(* Logix 5000 project; controller R1USB70001_CWRU_Scenario_Gen_20111116 vendor 1 type 14 code 54 rev 19.11; software revision 19.01; part 3 of 9 *)
(* tags used below, declared in another part *)
   DiscreteOutputsPv : DiscreteOutputsPv;
   EditScenarioPv : EditScenarioPv;
   CL_LP_B1_L1_SG1 : ALIAS FOR ACNR_CP_SG_N5:1:O.2;
   CL_LP_B1_L1_SG2 : ALIAS FOR ACNR_CP_SG_N5:1:O.3;
   CL_LP_B1_L2_SG1 : ALIAS FOR ACNR_CP_SG_N5:1:O.4;
   CL_LP_B1_L2_SG2 : ALIAS FOR ACNR_CP_SG_N5:1:O.5;
   CL_LP_B1_L3_SG1 : ALIAS FOR ACNR_CP_SG_N5:1:O.6;
   CL_LP_B1_L3_SG2 : ALIAS FOR ACNR_CP_SG_N5:1:O.7;
   CL_LP_B1_L4_SG1 : ALIAS FOR ACNR_CP_SG_N5:2:O.0;
   CL_LP_B1_L4_SG2 : ALIAS FOR ACNR_CP_SG_N5:2:O.1;
   CL_LP_B1_L5_SG1 : ALIAS FOR ACNR_CP_SG_N5:2:O.2;
   CL_LP_B1_L5_SG2 : ALIAS FOR ACNR_CP_SG_N5:2:O.3;
   CL_LP_B1_SG : ALIAS FOR ACNR_CP_SG_N5:1:O.1;
   CL_LP_B2_L1_SG1 : ALIAS FOR ACNR_CP_SG_N5:2:O.5;
   CL_LP_B2_L1_SG2 : ALIAS FOR ACNR_CP_SG_N5:2:O.6;
   CL_LP_B2_L2_SG1 : ALIAS FOR ACNR_CP_SG_N5:3:O.0;
   CL_LP_B2_L2_SG2 : ALIAS FOR ACNR_CP_SG_N5:3:O.1;
   CL_LP_B2_L3_SG1 : ALIAS FOR ACNR_CP_SG_N5:3:O.2;
   CL_LP_B2_L3_SG2 : ALIAS FOR ACNR_CP_SG_N5:3:O.3;
   CL_LP_B2_L4_SG1 : ALIAS FOR ACNR_CP_SG_N5:3:O.4;
   CL_LP_B2_L4_SG2 : ALIAS FOR ACNR_CP_SG_N5:3:O.5;
   CL_LP_B2_L5_SG1 : ALIAS FOR ACNR_CP_SG_N5:3:O.6;
   CL_LP_B2_L5_SG2 : ALIAS FOR ACNR_CP_SG_N5:3:O.7;
   CL_LP_B2_SG : ALIAS FOR ACNR_CP_SG_N5:2:O.4;
   CL_LP_ML_SG : ALIAS FOR ACNR_CP_SG_N5:1:O.0;
   EditScenario : EditScenarioPub;
   HMI : HMIPub;
   IL_LP_B1_L1_SG1 : ALIAS FOR ACNR_CP_SG_N5:4:O.2;
   IL_LP_B1_L1_SG2 : ALIAS FOR ACNR_CP_SG_N5:4:O.3;
   IL_LP_B1_L2_SG1 : ALIAS FOR ACNR_CP_SG_N5:4:O.4;
   IL_LP_B1_L2_SG2 : ALIAS FOR ACNR_CP_SG_N5:4:O.5;
   IL_LP_B1_L3_SG1 : ALIAS FOR ACNR_CP_SG_N5:4:O.6;
   IL_LP_B1_L3_SG2 : ALIAS FOR ACNR_CP_SG_N5:4:O.7;
   IL_LP_B1_L4_SG1 : ALIAS FOR ACNR_CP_SG_N5:5:O.0;
   IL_LP_B1_L4_SG2 : ALIAS FOR ACNR_CP_SG_N5:5:O.1;
   IL_LP_B1_L5_SG1 : ALIAS FOR ACNR_CP_SG_N5:5:O.2;
   IL_LP_B1_L5_SG2 : ALIAS FOR ACNR_CP_SG_N5:5:O.3;
   IL_LP_B1_SG : ALIAS FOR ACNR_CP_SG_N5:4:O.1;
   IL_LP_B2_L1_SG1 : ALIAS FOR ACNR_CP_SG_N5:5:O.5;
   IL_LP_B2_L1_SG2 : ALIAS FOR ACNR_CP_SG_N5:5:O.6;
   IL_LP_B2_L2_SG1 : ALIAS FOR ACNR_CP_SG_N5:6:O.0;
   IL_LP_B2_L2_SG2 : ALIAS FOR ACNR_CP_SG_N5:6:O.1;
   IL_LP_B2_L3_SG1 : ALIAS FOR ACNR_CP_SG_N5:6:O.2;
   IL_LP_B2_L3_SG2 : ALIAS FOR ACNR_CP_SG_N5:6:O.3;
   IL_LP_B2_L4_SG1 : ALIAS FOR ACNR_CP_SG_N5:6:O.4;
   IL_LP_B2_L4_SG2 : ALIAS FOR ACNR_CP_SG_N5:6:O.5;
   IL_LP_B2_L5_SG1 : ALIAS FOR ACNR_CP_SG_N5:6:O.6;
   IL_LP_B2_L5_SG2 : ALIAS FOR ACNR_CP_SG_N5:6:O.7;
   IL_LP_B2_SG : ALIAS FOR ACNR_CP_SG_N5:5:O.4;
   IL_LP_ML_SG : ALIAS FOR ACNR_CP_SG_N5:4:O.0;
   RL_LP_B1_L5_SG2 : ALIAS FOR ACNR_RP_SG_N4:2:O.3;
   RL_LP_B2_L1_SG1 : ALIAS FOR ACNR_RP_SG_N4:2:O.5;
   RL_LP_B2_L1_SG2 : ALIAS FOR ACNR_RP_SG_N4:2:O.6;
   RL_LP_B2_L2_SG1 : ALIAS FOR ACNR_RP_SG_N4:2:O.7;
   RL_LP_B2_L2_SG2 : ALIAS FOR ACNR_RP_SG_N4:3:O.0;
   RL_LP_B2_L3_SG1 : ALIAS FOR ACNR_RP_SG_N4:3:O.1;
   RL_LP_B2_L3_SG2 : ALIAS FOR ACNR_RP_SG_N4:3:O.2;
   RL_LP_B2_L4_SG1 : ALIAS FOR ACNR_RP_SG_N4:3:O.3;
   RL_LP_B2_L4_SG2 : ALIAS FOR ACNR_RP_SG_N4:3:O.4;
   RL_LP_B2_L5_SG1 : ALIAS FOR ACNR_RP_SG_N4:3:O.5;
   RL_LP_B2_L5_SG2 : ALIAS FOR ACNR_RP_SG_N4:3:O.6;
   RL_LP_B2_SG : ALIAS FOR ACNR_RP_SG_N4:2:O.4;
   RL_LP_B3_L1_SG1 : ALIAS FOR ACNR_RP_SG_N4:4:O.0;
   RL_LP_B3_L1_SG2 : ALIAS FOR ACNR_RP_SG_N4:4:O.1;
   RL_LP_B3_L2_SG1 : ALIAS FOR ACNR_RP_SG_N4:4:O.2;
   RL_LP_B3_L2_SG2 : ALIAS FOR ACNR_RP_SG_N4:4:O.3;
   RL_LP_B3_L3_SG1 : ALIAS FOR ACNR_RP_SG_N4:4:O.4;
   RL_LP_B3_L3_SG2 : ALIAS FOR ACNR_RP_SG_N4:4:O.5;
   RL_LP_B3_L4_SG1 : ALIAS FOR ACNR_RP_SG_N4:4:O.6;
   RL_LP_B3_L4_SG2 : ALIAS FOR ACNR_RP_SG_N4:4:O.7;
   RL_LP_B3_L5_SG1 : ALIAS FOR ACNR_RP_SG_N4:5:O.0;
   RL_LP_B3_L5_SG2 : ALIAS FOR ACNR_RP_SG_N4:5:O.1;
   RL_LP_B3_SG : ALIAS FOR ACNR_RP_SG_N4:3:O.7;
   RL_LP_B4_L1_SG1 : ALIAS FOR ACNR_RP_SG_N4:5:O.3;
   RL_LP_B4_L1_SG2 : ALIAS FOR ACNR_RP_SG_N4:5:O.4;
   RL_LP_B4_L2_SG1 : ALIAS FOR ACNR_RP_SG_N4:5:O.5;
   RL_LP_B4_L2_SG2 : ALIAS FOR ACNR_RP_SG_N4:5:O.6;
   RL_LP_B4_L3_SG1 : ALIAS FOR ACNR_RP_SG_N4:5:O.7;
   RL_LP_B4_L3_SG2 : ALIAS FOR ACNR_RP_SG_N4:6:O.0;
   RL_LP_B4_L4_SG1 : ALIAS FOR ACNR_RP_SG_N4:6:O.1;
   RL_LP_B4_L4_SG2 : ALIAS FOR ACNR_RP_SG_N4:6:O.2;
   RL_LP_B4_L5_SG1 : ALIAS FOR ACNR_RP_SG_N4:6:O.3;
   RL_LP_B4_L5_SG2 : ALIAS FOR ACNR_RP_SG_N4:6:O.4;
   RL_LP_B4_SG : ALIAS FOR ACNR_RP_SG_N4:5:O.2;
   Scenario : Scenario_Def[100];
(* MainProgram, continued *)

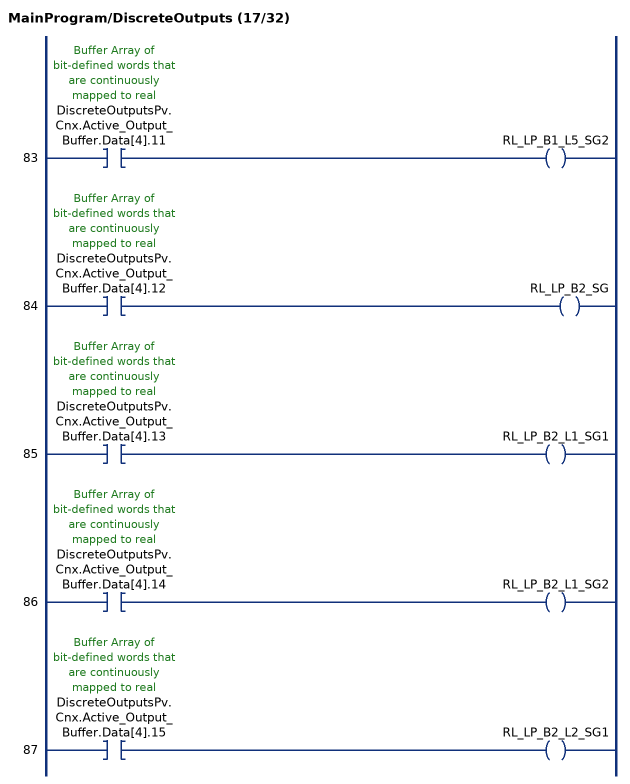
   83: XIC(DiscreteOutputsPv.Cnx.Active_Output_Buffer.Data[4].11)OTE(RL_LP_B1_L5_SG2);
   84: XIC(DiscreteOutputsPv.Cnx.Active_Output_Buffer.Data[4].12)OTE(RL_LP_B2_SG);
   85: XIC(DiscreteOutputsPv.Cnx.Active_Output_Buffer.Data[4].13)OTE(RL_LP_B2_L1_SG1);
   86: XIC(DiscreteOutputsPv.Cnx.Active_Output_Buffer.Data[4].14)OTE(RL_LP_B2_L1_SG2);
   87: XIC(DiscreteOutputsPv.Cnx.Active_Output_Buffer.Data[4].15)OTE(RL_LP_B2_L2_SG1);
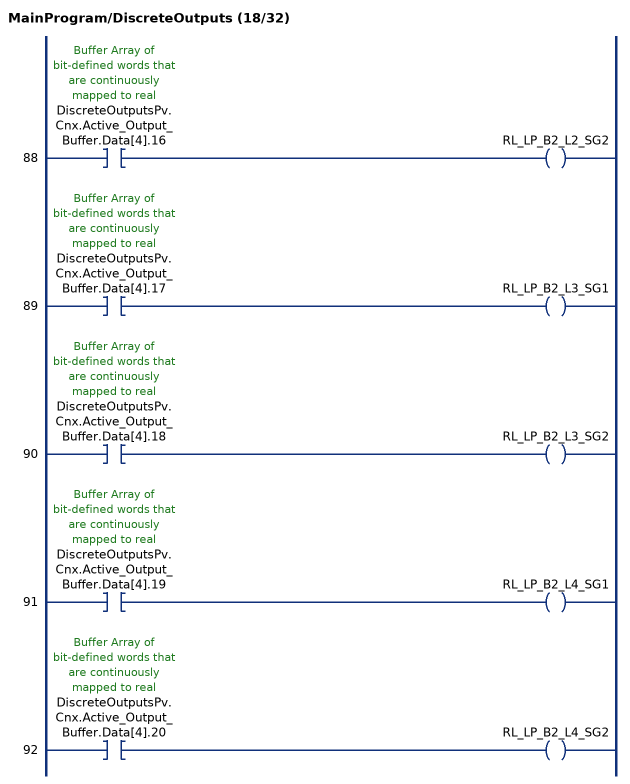
   88: XIC(DiscreteOutputsPv.Cnx.Active_Output_Buffer.Data[4].16)OTE(RL_LP_B2_L2_SG2);
   89: XIC(DiscreteOutputsPv.Cnx.Active_Output_Buffer.Data[4].17)OTE(RL_LP_B2_L3_SG1);
   90: XIC(DiscreteOutputsPv.Cnx.Active_Output_Buffer.Data[4].18)OTE(RL_LP_B2_L3_SG2);
   91: XIC(DiscreteOutputsPv.Cnx.Active_Output_Buffer.Data[4].19)OTE(RL_LP_B2_L4_SG1);
   92: XIC(DiscreteOutputsPv.Cnx.Active_Output_Buffer.Data[4].20)OTE(RL_LP_B2_L4_SG2);
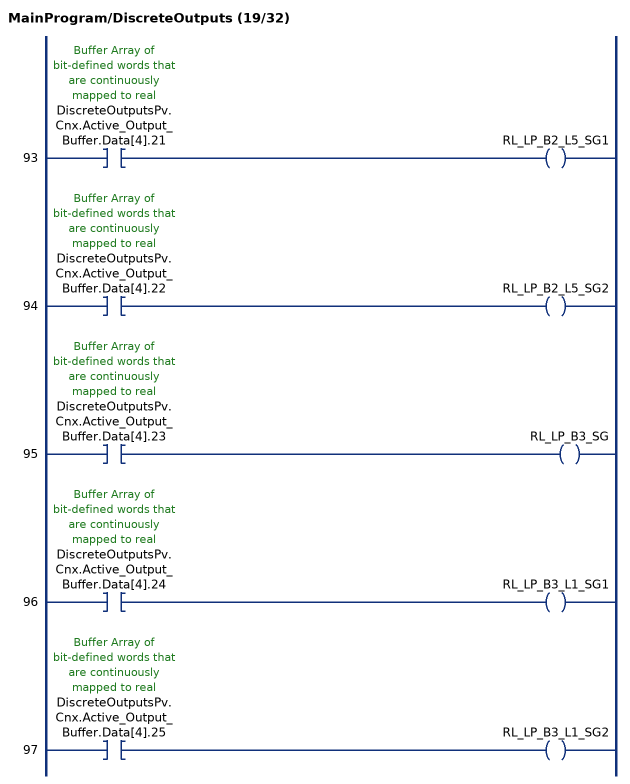
   93: XIC(DiscreteOutputsPv.Cnx.Active_Output_Buffer.Data[4].21)OTE(RL_LP_B2_L5_SG1);
   94: XIC(DiscreteOutputsPv.Cnx.Active_Output_Buffer.Data[4].22)OTE(RL_LP_B2_L5_SG2);
   95: XIC(DiscreteOutputsPv.Cnx.Active_Output_Buffer.Data[4].23)OTE(RL_LP_B3_SG);
   96: XIC(DiscreteOutputsPv.Cnx.Active_Output_Buffer.Data[4].24)OTE(RL_LP_B3_L1_SG1);
   97: XIC(DiscreteOutputsPv.Cnx.Active_Output_Buffer.Data[4].25)OTE(RL_LP_B3_L1_SG2);
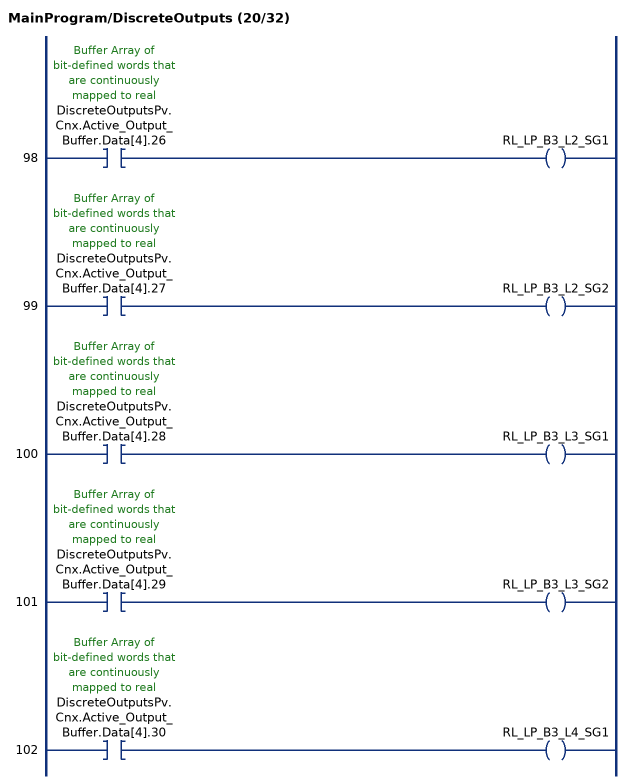
   98: XIC(DiscreteOutputsPv.Cnx.Active_Output_Buffer.Data[4].26)OTE(RL_LP_B3_L2_SG1);
   99: XIC(DiscreteOutputsPv.Cnx.Active_Output_Buffer.Data[4].27)OTE(RL_LP_B3_L2_SG2);
   100: XIC(DiscreteOutputsPv.Cnx.Active_Output_Buffer.Data[4].28)OTE(RL_LP_B3_L3_SG1);
   101: XIC(DiscreteOutputsPv.Cnx.Active_Output_Buffer.Data[4].29)OTE(RL_LP_B3_L3_SG2);
   102: XIC(DiscreteOutputsPv.Cnx.Active_Output_Buffer.Data[4].30)OTE(RL_LP_B3_L4_SG1);
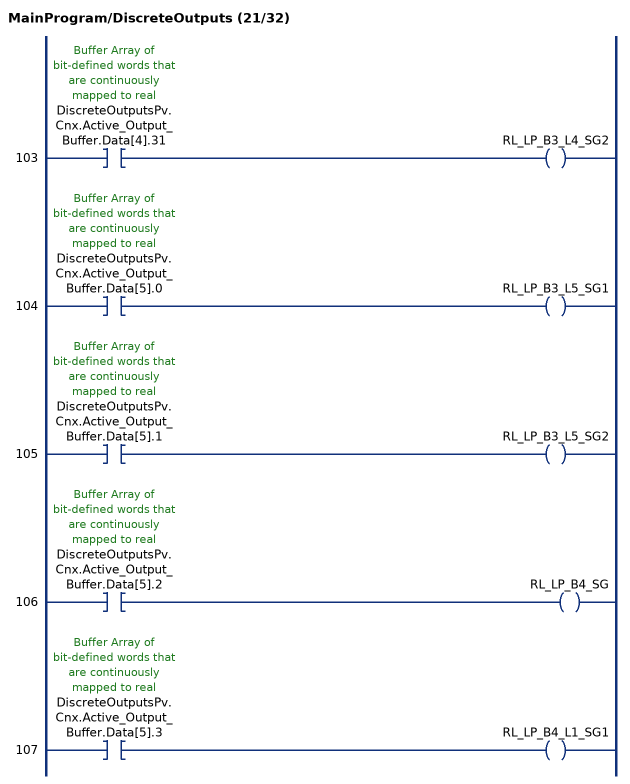
   103: XIC(DiscreteOutputsPv.Cnx.Active_Output_Buffer.Data[4].31)OTE(RL_LP_B3_L4_SG2);
   104: XIC(DiscreteOutputsPv.Cnx.Active_Output_Buffer.Data[5].0)OTE(RL_LP_B3_L5_SG1);
   105: XIC(DiscreteOutputsPv.Cnx.Active_Output_Buffer.Data[5].1)OTE(RL_LP_B3_L5_SG2);
   106: XIC(DiscreteOutputsPv.Cnx.Active_Output_Buffer.Data[5].2)OTE(RL_LP_B4_SG);
   107: XIC(DiscreteOutputsPv.Cnx.Active_Output_Buffer.Data[5].3)OTE(RL_LP_B4_L1_SG1);
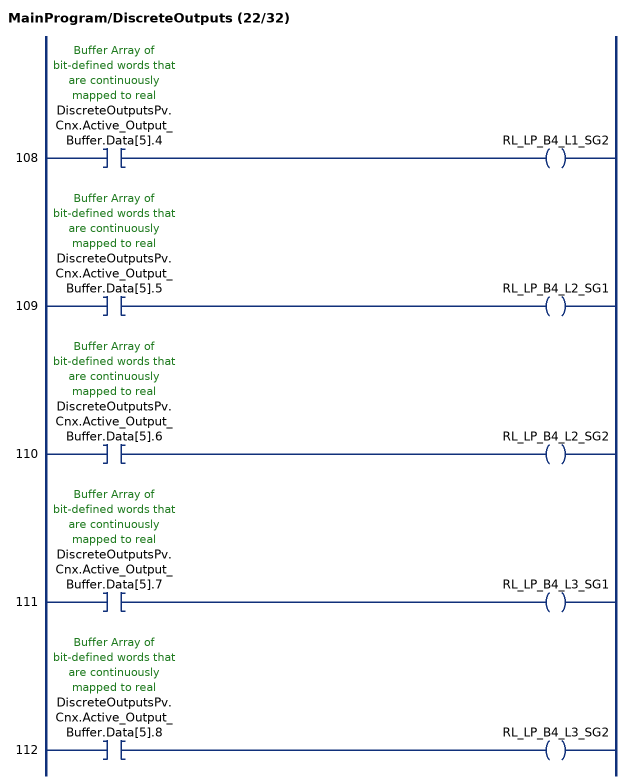
   108: XIC(DiscreteOutputsPv.Cnx.Active_Output_Buffer.Data[5].4)OTE(RL_LP_B4_L1_SG2);
   109: XIC(DiscreteOutputsPv.Cnx.Active_Output_Buffer.Data[5].5)OTE(RL_LP_B4_L2_SG1);
   110: XIC(DiscreteOutputsPv.Cnx.Active_Output_Buffer.Data[5].6)OTE(RL_LP_B4_L2_SG2);
   111: XIC(DiscreteOutputsPv.Cnx.Active_Output_Buffer.Data[5].7)OTE(RL_LP_B4_L3_SG1);
   112: XIC(DiscreteOutputsPv.Cnx.Active_Output_Buffer.Data[5].8)OTE(RL_LP_B4_L3_SG2);
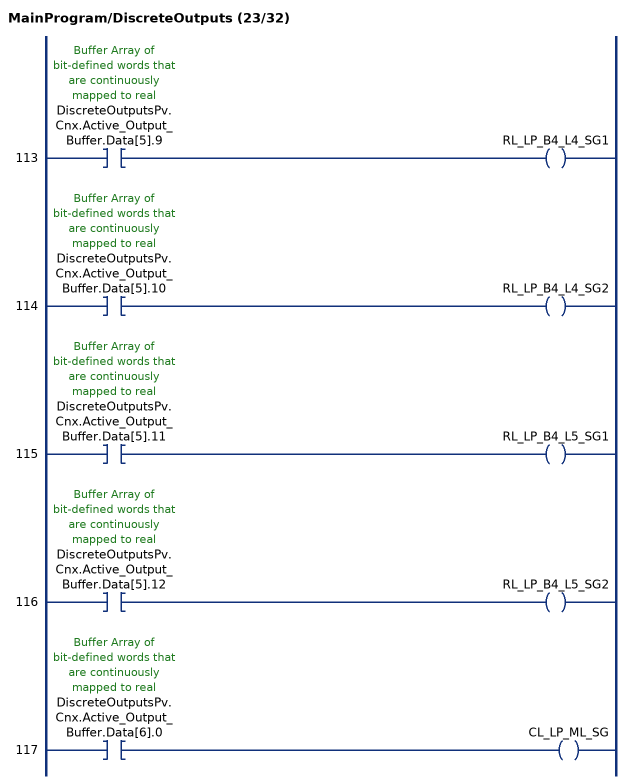
   113: XIC(DiscreteOutputsPv.Cnx.Active_Output_Buffer.Data[5].9)OTE(RL_LP_B4_L4_SG1);
   114: XIC(DiscreteOutputsPv.Cnx.Active_Output_Buffer.Data[5].10)OTE(RL_LP_B4_L4_SG2);
   115: XIC(DiscreteOutputsPv.Cnx.Active_Output_Buffer.Data[5].11)OTE(RL_LP_B4_L5_SG1);
   116: XIC(DiscreteOutputsPv.Cnx.Active_Output_Buffer.Data[5].12)OTE(RL_LP_B4_L5_SG2);
   117: XIC(DiscreteOutputsPv.Cnx.Active_Output_Buffer.Data[6].0)OTE(CL_LP_ML_SG);
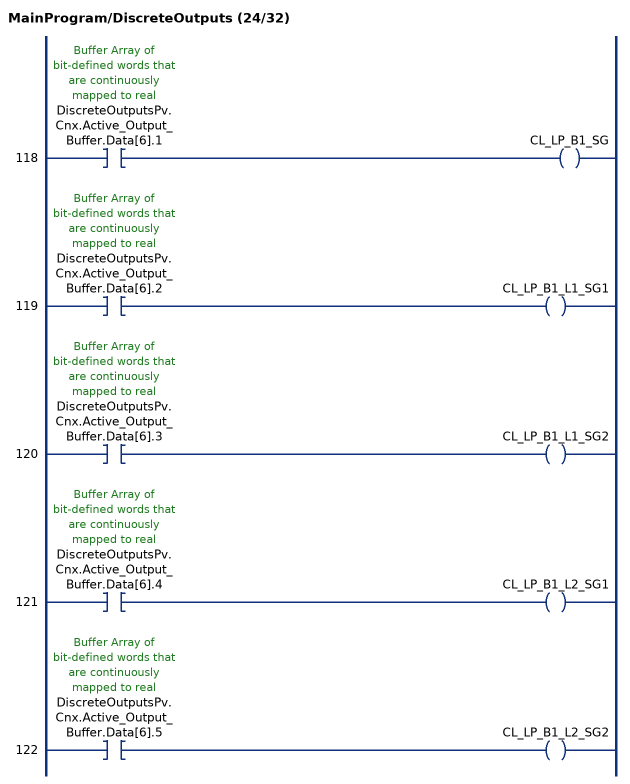
   118: XIC(DiscreteOutputsPv.Cnx.Active_Output_Buffer.Data[6].1)OTE(CL_LP_B1_SG);
   119: XIC(DiscreteOutputsPv.Cnx.Active_Output_Buffer.Data[6].2)OTE(CL_LP_B1_L1_SG1);
   120: XIC(DiscreteOutputsPv.Cnx.Active_Output_Buffer.Data[6].3)OTE(CL_LP_B1_L1_SG2);
   121: XIC(DiscreteOutputsPv.Cnx.Active_Output_Buffer.Data[6].4)OTE(CL_LP_B1_L2_SG1);
   122: XIC(DiscreteOutputsPv.Cnx.Active_Output_Buffer.Data[6].5)OTE(CL_LP_B1_L2_SG2);
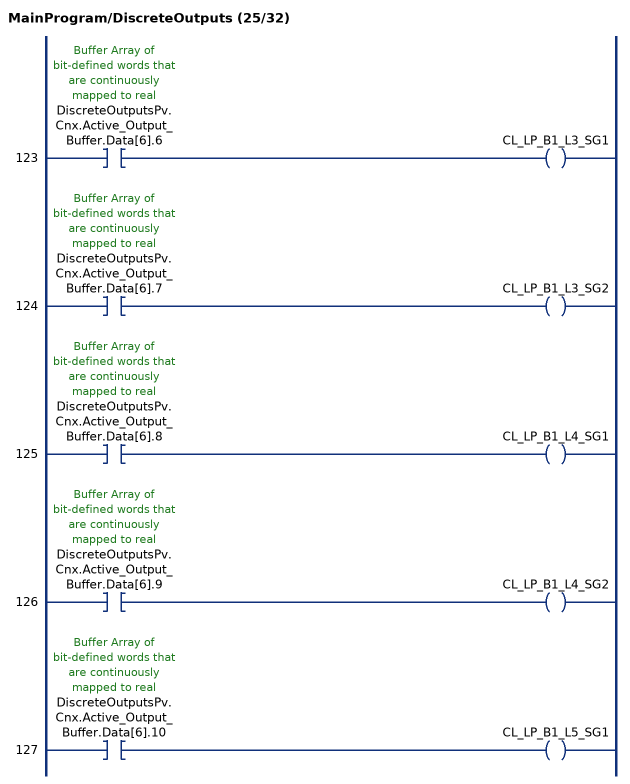
   123: XIC(DiscreteOutputsPv.Cnx.Active_Output_Buffer.Data[6].6)OTE(CL_LP_B1_L3_SG1);
   124: XIC(DiscreteOutputsPv.Cnx.Active_Output_Buffer.Data[6].7)OTE(CL_LP_B1_L3_SG2);
   125: XIC(DiscreteOutputsPv.Cnx.Active_Output_Buffer.Data[6].8)OTE(CL_LP_B1_L4_SG1);
   126: XIC(DiscreteOutputsPv.Cnx.Active_Output_Buffer.Data[6].9)OTE(CL_LP_B1_L4_SG2);
   127: XIC(DiscreteOutputsPv.Cnx.Active_Output_Buffer.Data[6].10)OTE(CL_LP_B1_L5_SG1);
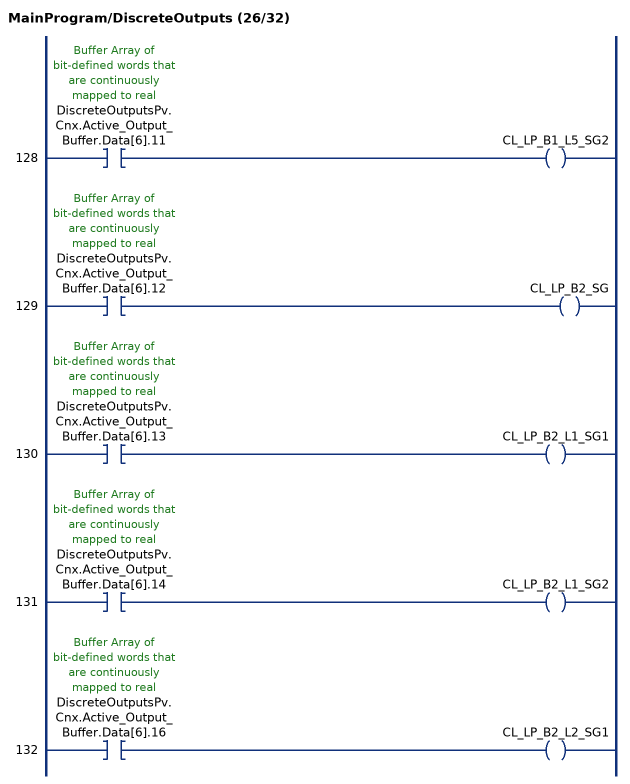
   128: XIC(DiscreteOutputsPv.Cnx.Active_Output_Buffer.Data[6].11)OTE(CL_LP_B1_L5_SG2);
   129: XIC(DiscreteOutputsPv.Cnx.Active_Output_Buffer.Data[6].12)OTE(CL_LP_B2_SG);
   130: XIC(DiscreteOutputsPv.Cnx.Active_Output_Buffer.Data[6].13)OTE(CL_LP_B2_L1_SG1);
   131: XIC(DiscreteOutputsPv.Cnx.Active_Output_Buffer.Data[6].14)OTE(CL_LP_B2_L1_SG2);
   132: XIC(DiscreteOutputsPv.Cnx.Active_Output_Buffer.Data[6].16)OTE(CL_LP_B2_L2_SG1);
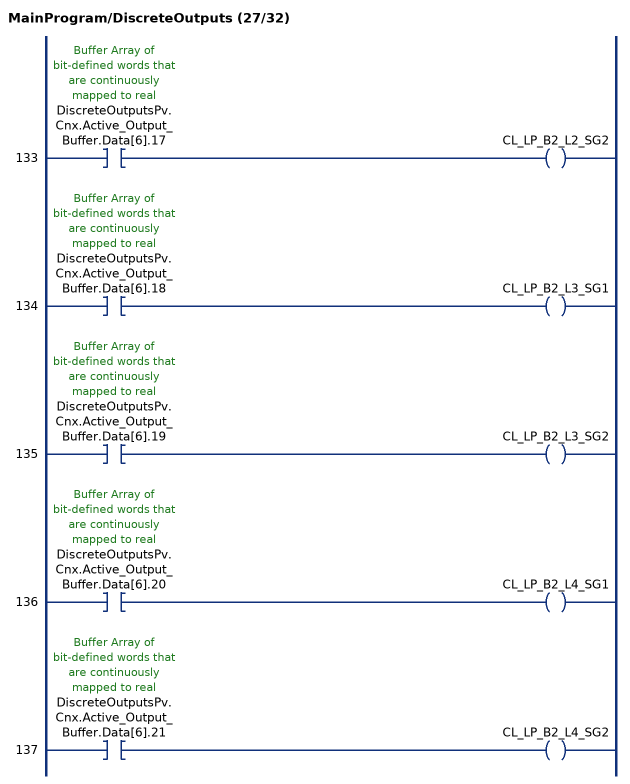
   133: XIC(DiscreteOutputsPv.Cnx.Active_Output_Buffer.Data[6].17)OTE(CL_LP_B2_L2_SG2);
   134: XIC(DiscreteOutputsPv.Cnx.Active_Output_Buffer.Data[6].18)OTE(CL_LP_B2_L3_SG1);
   135: XIC(DiscreteOutputsPv.Cnx.Active_Output_Buffer.Data[6].19)OTE(CL_LP_B2_L3_SG2);
   136: XIC(DiscreteOutputsPv.Cnx.Active_Output_Buffer.Data[6].20)OTE(CL_LP_B2_L4_SG1);
   137: XIC(DiscreteOutputsPv.Cnx.Active_Output_Buffer.Data[6].21)OTE(CL_LP_B2_L4_SG2);
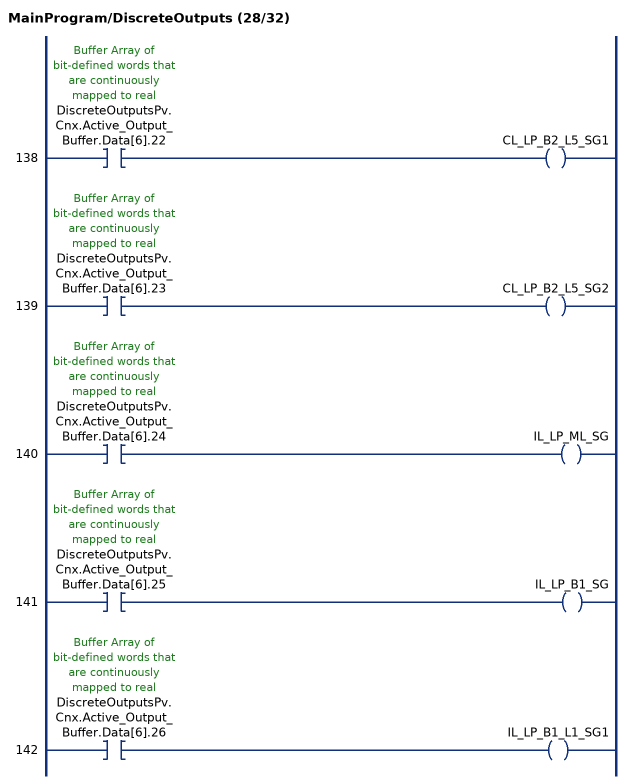
   138: XIC(DiscreteOutputsPv.Cnx.Active_Output_Buffer.Data[6].22)OTE(CL_LP_B2_L5_SG1);
   139: XIC(DiscreteOutputsPv.Cnx.Active_Output_Buffer.Data[6].23)OTE(CL_LP_B2_L5_SG2);
   140: XIC(DiscreteOutputsPv.Cnx.Active_Output_Buffer.Data[6].24)OTE(IL_LP_ML_SG);
   141: XIC(DiscreteOutputsPv.Cnx.Active_Output_Buffer.Data[6].25)OTE(IL_LP_B1_SG);
   142: XIC(DiscreteOutputsPv.Cnx.Active_Output_Buffer.Data[6].26)OTE(IL_LP_B1_L1_SG1);
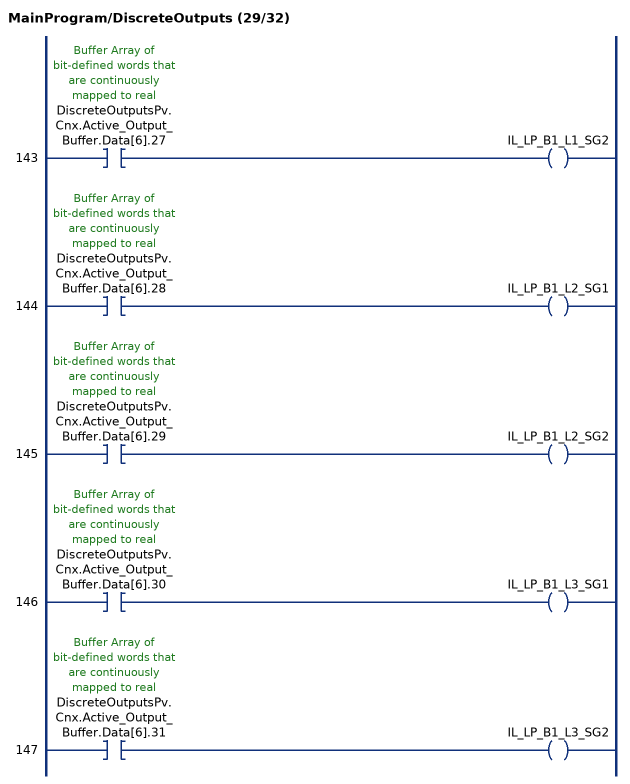
   143: XIC(DiscreteOutputsPv.Cnx.Active_Output_Buffer.Data[6].27)OTE(IL_LP_B1_L1_SG2);
   144: XIC(DiscreteOutputsPv.Cnx.Active_Output_Buffer.Data[6].28)OTE(IL_LP_B1_L2_SG1);
   145: XIC(DiscreteOutputsPv.Cnx.Active_Output_Buffer.Data[6].29)OTE(IL_LP_B1_L2_SG2);
   146: XIC(DiscreteOutputsPv.Cnx.Active_Output_Buffer.Data[6].30)OTE(IL_LP_B1_L3_SG1);
   147: XIC(DiscreteOutputsPv.Cnx.Active_Output_Buffer.Data[6].31)OTE(IL_LP_B1_L3_SG2);
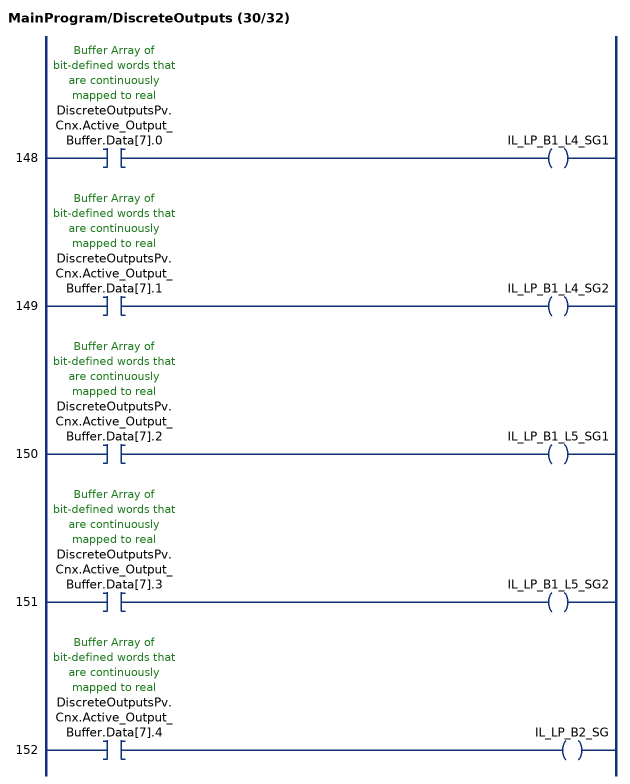
   148: XIC(DiscreteOutputsPv.Cnx.Active_Output_Buffer.Data[7].0)OTE(IL_LP_B1_L4_SG1);
   149: XIC(DiscreteOutputsPv.Cnx.Active_Output_Buffer.Data[7].1)OTE(IL_LP_B1_L4_SG2);
   150: XIC(DiscreteOutputsPv.Cnx.Active_Output_Buffer.Data[7].2)OTE(IL_LP_B1_L5_SG1);
   151: XIC(DiscreteOutputsPv.Cnx.Active_Output_Buffer.Data[7].3)OTE(IL_LP_B1_L5_SG2);
   152: XIC(DiscreteOutputsPv.Cnx.Active_Output_Buffer.Data[7].4)OTE(IL_LP_B2_SG);
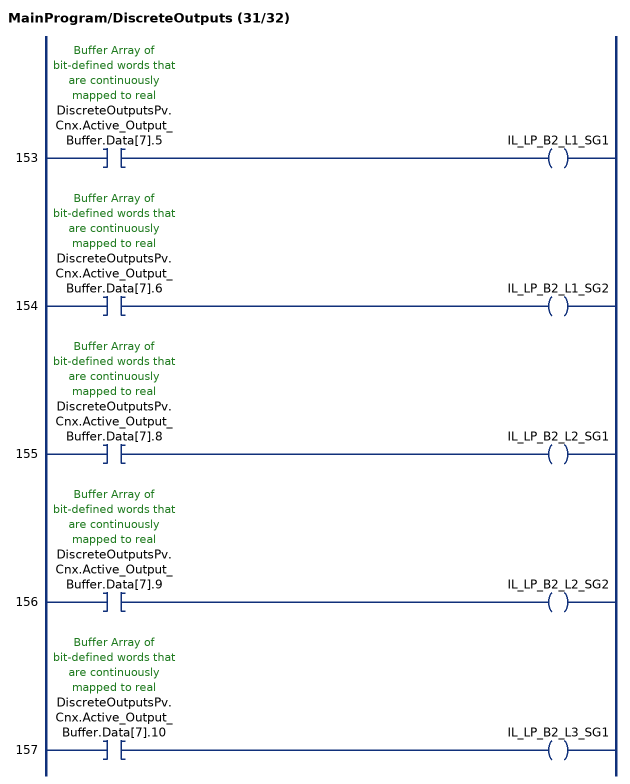
   153: XIC(DiscreteOutputsPv.Cnx.Active_Output_Buffer.Data[7].5)OTE(IL_LP_B2_L1_SG1);
   154: XIC(DiscreteOutputsPv.Cnx.Active_Output_Buffer.Data[7].6)OTE(IL_LP_B2_L1_SG2);
   155: XIC(DiscreteOutputsPv.Cnx.Active_Output_Buffer.Data[7].8)OTE(IL_LP_B2_L2_SG1);
   156: XIC(DiscreteOutputsPv.Cnx.Active_Output_Buffer.Data[7].9)OTE(IL_LP_B2_L2_SG2);
   157: XIC(DiscreteOutputsPv.Cnx.Active_Output_Buffer.Data[7].10)OTE(IL_LP_B2_L3_SG1);
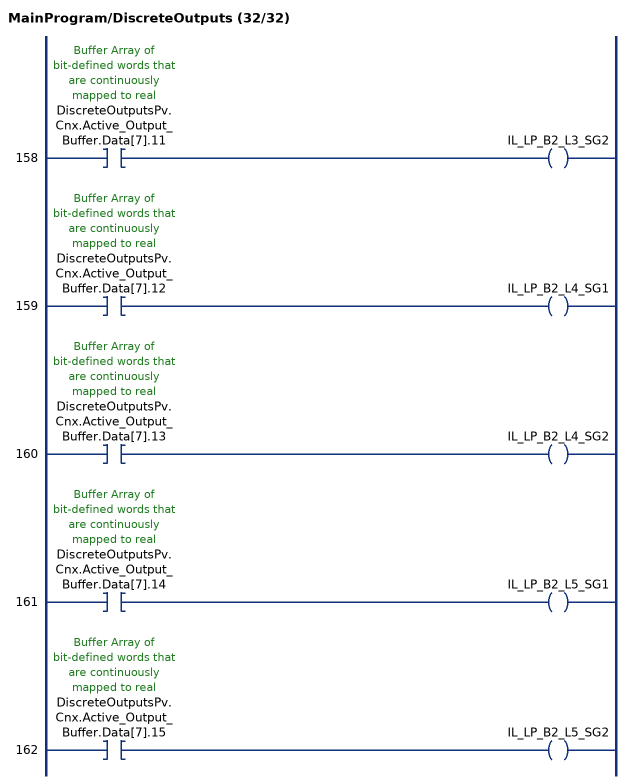
   158: XIC(DiscreteOutputsPv.Cnx.Active_Output_Buffer.Data[7].11)OTE(IL_LP_B2_L3_SG2);
   159: XIC(DiscreteOutputsPv.Cnx.Active_Output_Buffer.Data[7].12)OTE(IL_LP_B2_L4_SG1);
   160: XIC(DiscreteOutputsPv.Cnx.Active_Output_Buffer.Data[7].13)OTE(IL_LP_B2_L4_SG2);
   161: XIC(DiscreteOutputsPv.Cnx.Active_Output_Buffer.Data[7].14)OTE(IL_LP_B2_L5_SG1);
   162: XIC(DiscreteOutputsPv.Cnx.Active_Output_Buffer.Data[7].15)OTE(IL_LP_B2_L5_SG2);
END_ROUTINE

ROUTINE EditScenario   (* ladder *)
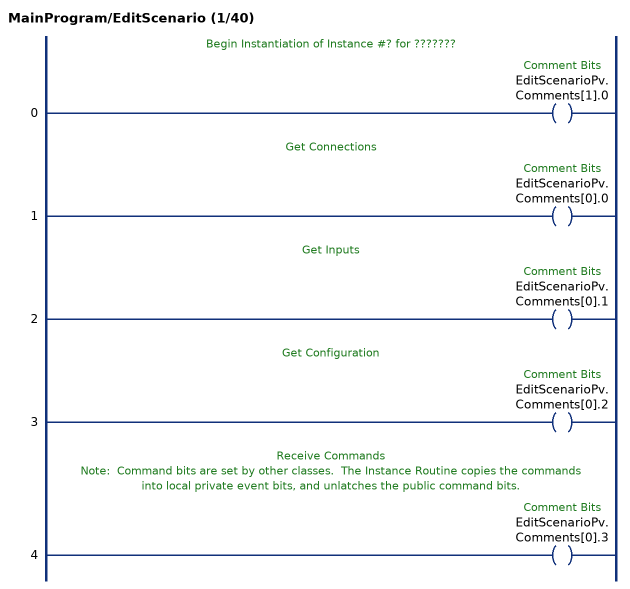
   // Begin Instantiation of Instance #? for ???????
   0: OTE(EditScenarioPv.Comments[1].0);
   // Get Connections
   1: OTE(EditScenarioPv.Comments[0].0);
   // Get Inputs
   2: OTE(EditScenarioPv.Comments[0].1);
   // Get Configuration
   3: OTE(EditScenarioPv.Comments[0].2);
   // Receive Commands
   // Note:  Command bits are set by other classes.  The Instance Routine copies the commands into local private event bits, and unlatches the public command bits.
   4: OTE(EditScenarioPv.Comments[0].3);
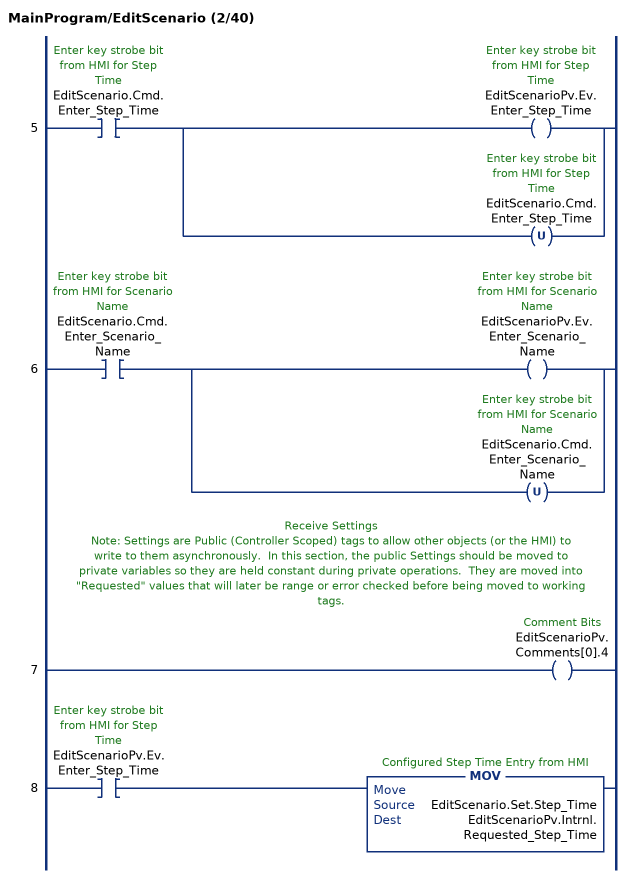
   5: XIC(EditScenario.Cmd.Enter_Step_Time)[OTE(EditScenarioPv.Ev.Enter_Step_Time) ,OTU(EditScenario.Cmd.Enter_Step_Time) ];
   6: XIC(EditScenario.Cmd.Enter_Scenario_Name)[OTE(EditScenarioPv.Ev.Enter_Scenario_Name) ,OTU(EditScenario.Cmd.Enter_Scenario_Name) ];
   // Receive Settings
   // Note: Settings are Public (Controller Scoped) tags to allow other objects (or the HMI) to write to them asynchronously.  In this section, the public Settings should be moved to private variables so they are held constant during private operations.  They are moved into "Requested" values that will later be range or error checked before being moved to working tags.
   7: OTE(EditScenarioPv.Comments[0].4);
   8: XIC(EditScenarioPv.Ev.Enter_Step_Time)MOV(EditScenario.Set.Step_Time,EditScenarioPv.Intrnl.Requested_Step_Time);
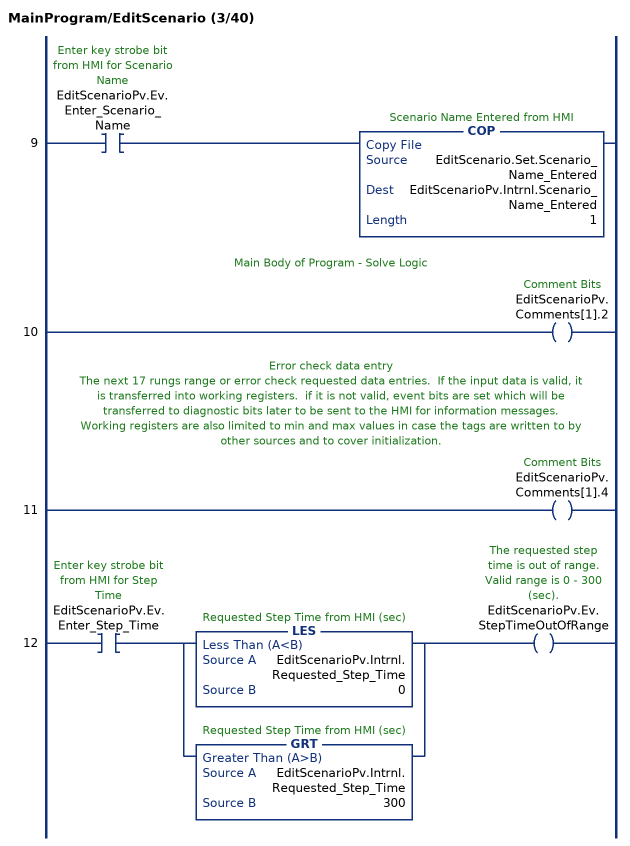
   9: XIC(EditScenarioPv.Ev.Enter_Scenario_Name)COP(EditScenario.Set.Scenario_Name_Entered,EditScenarioPv.Intrnl.Scenario_Name_Entered,1);
   // Main Body of Program - Solve Logic
   10: OTE(EditScenarioPv.Comments[1].2);
   // Error check data entry
   // The next 17 rungs range or error check requested data entries.  If the input data is valid, it is transferred into working registers.  if it is not valid, event bits are set which will be transferred to diagnostic bits later to be sent to the HMI for information messages.
   // Working registers are also limited to min and max values in case the tags are written to by other sources and to cover initialization.
   11: OTE(EditScenarioPv.Comments[1].4);
   12: XIC(EditScenarioPv.Ev.Enter_Step_Time)[LES(EditScenarioPv.Intrnl.Requested_Step_Time,0) ,GRT(EditScenarioPv.Intrnl.Requested_Step_Time,300) ]OTE(EditScenarioPv.Ev.StepTimeOutOfRange);
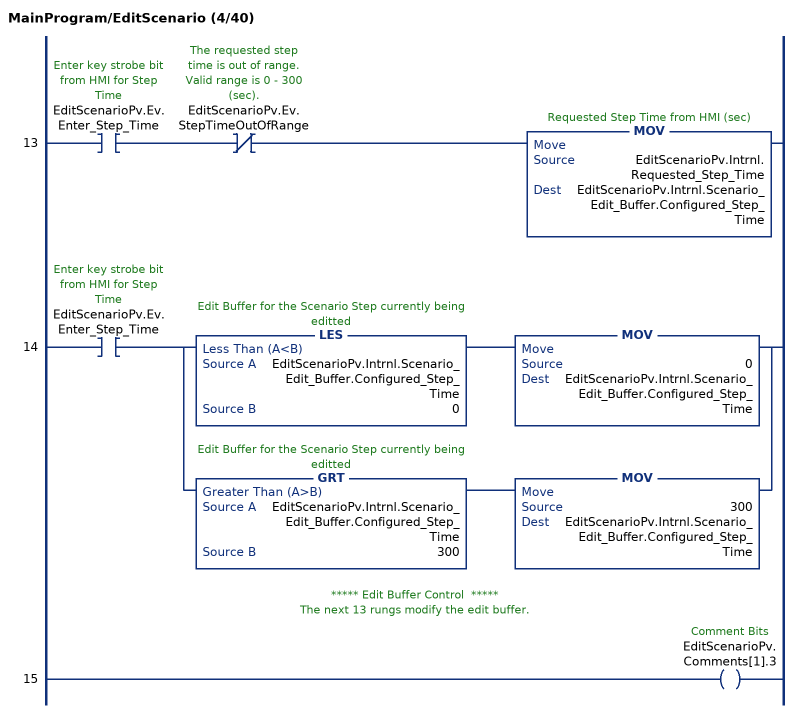
   13: XIC(EditScenarioPv.Ev.Enter_Step_Time)XIO(EditScenarioPv.Ev.StepTimeOutOfRange)MOV(EditScenarioPv.Intrnl.Requested_Step_Time,EditScenarioPv.Intrnl.Scenario_Edit_Buffer.Configured_Step_Time);
   14: XIC(EditScenarioPv.Ev.Enter_Step_Time)[LES(EditScenarioPv.Intrnl.Scenario_Edit_Buffer.Configured_Step_Time,0) MOV(0,EditScenarioPv.Intrnl.Scenario_Edit_Buffer.Configured_Step_Time) ,GRT(EditScenarioPv.Intrnl.Scenario_Edit_Buffer.Configured_Step_Time,300) MOV(300,EditScenarioPv.Intrnl.Scenario_Edit_Buffer.Configured_Step_Time) ];
   // ***** Edit Buffer Control  *****
   // The next 13 rungs modify the edit buffer.
   15: OTE(EditScenarioPv.Comments[1].3);
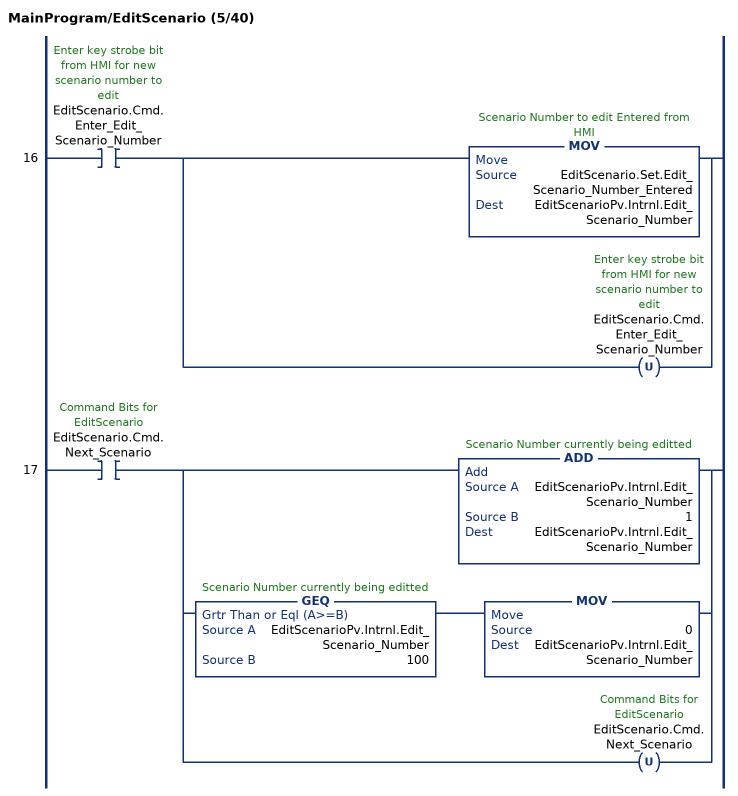
   16: XIC(EditScenario.Cmd.Enter_Edit_Scenario_Number)[MOV(EditScenario.Set.Edit_Scenario_Number_Entered,EditScenarioPv.Intrnl.Edit_Scenario_Number) ,OTU(EditScenario.Cmd.Enter_Edit_Scenario_Number) ];
   17: XIC(EditScenario.Cmd.Next_Scenario)[ADD(EditScenarioPv.Intrnl.Edit_Scenario_Number,1,EditScenarioPv.Intrnl.Edit_Scenario_Number) ,GEQ(EditScenarioPv.Intrnl.Edit_Scenario_Number,100) MOV(0,EditScenarioPv.Intrnl.Edit_Scenario_Number) ,OTU(EditScenario.Cmd.Next_Scenario) ];
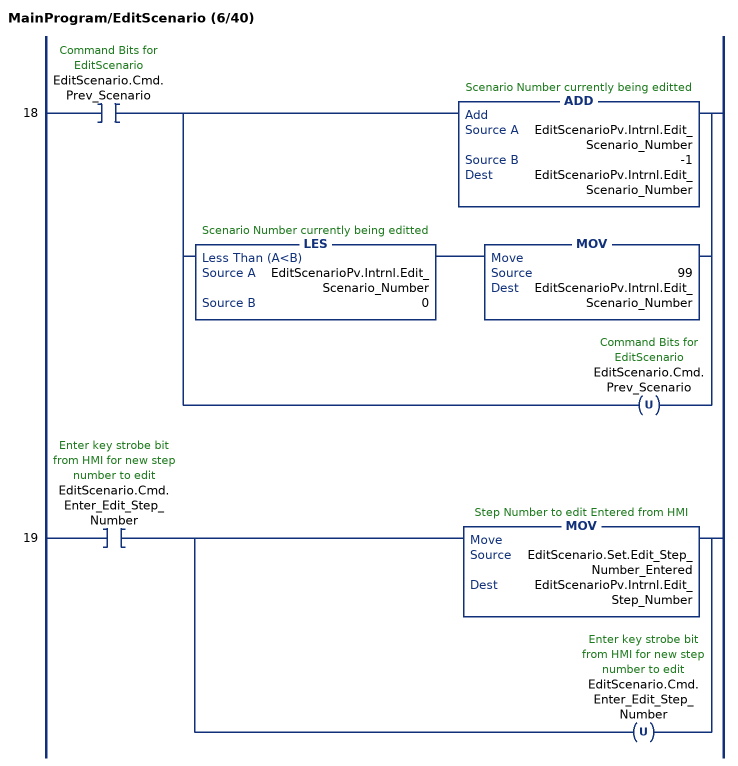
   18: XIC(EditScenario.Cmd.Prev_Scenario)[ADD(EditScenarioPv.Intrnl.Edit_Scenario_Number,-1,EditScenarioPv.Intrnl.Edit_Scenario_Number) ,LES(EditScenarioPv.Intrnl.Edit_Scenario_Number,0) MOV(99,EditScenarioPv.Intrnl.Edit_Scenario_Number) ,OTU(EditScenario.Cmd.Prev_Scenario) ];
   19: XIC(EditScenario.Cmd.Enter_Edit_Step_Number)[MOV(EditScenario.Set.Edit_Step_Number_Entered,EditScenarioPv.Intrnl.Edit_Step_Number) ,OTU(EditScenario.Cmd.Enter_Edit_Step_Number) ];
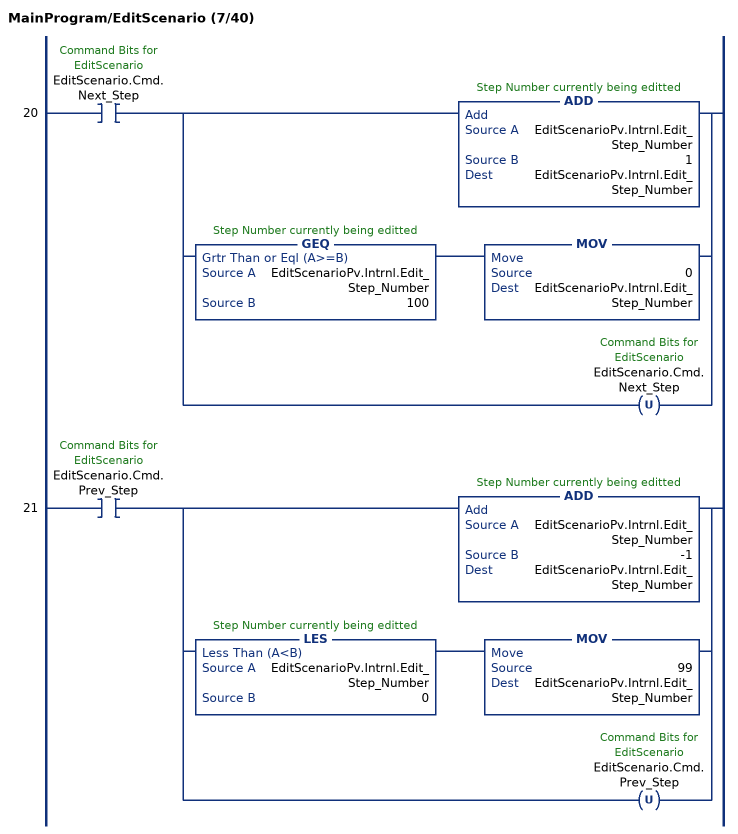
   20: XIC(EditScenario.Cmd.Next_Step)[ADD(EditScenarioPv.Intrnl.Edit_Step_Number,1,EditScenarioPv.Intrnl.Edit_Step_Number) ,GEQ(EditScenarioPv.Intrnl.Edit_Step_Number,100) MOV(0,EditScenarioPv.Intrnl.Edit_Step_Number) ,OTU(EditScenario.Cmd.Next_Step) ];
   21: XIC(EditScenario.Cmd.Prev_Step)[ADD(EditScenarioPv.Intrnl.Edit_Step_Number,-1,EditScenarioPv.Intrnl.Edit_Step_Number) ,LES(EditScenarioPv.Intrnl.Edit_Step_Number,0) MOV(99,EditScenarioPv.Intrnl.Edit_Step_Number) ,OTU(EditScenario.Cmd.Prev_Step) ];
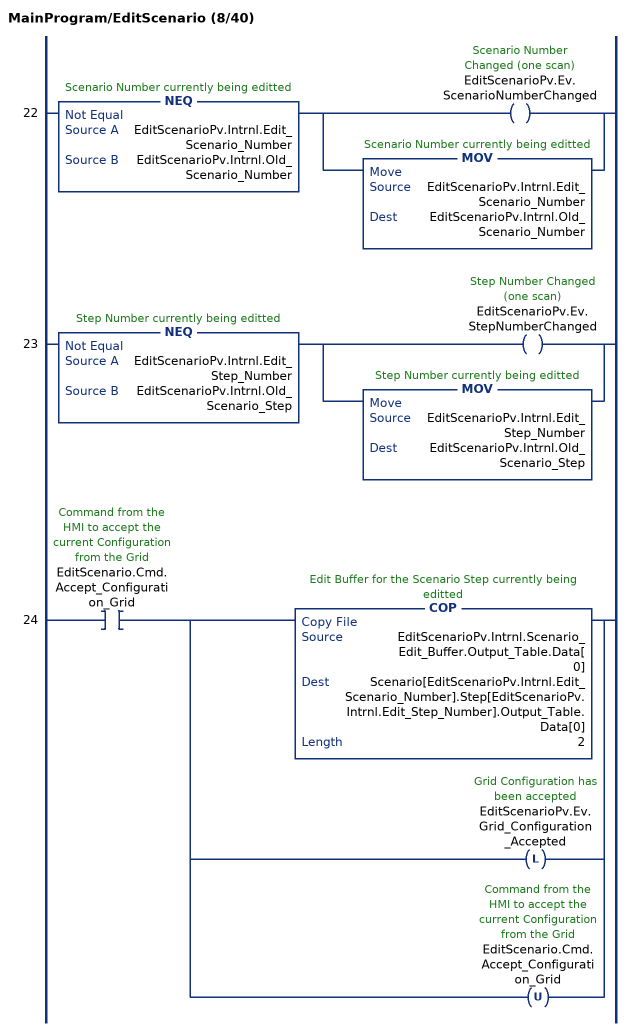
   22: NEQ(EditScenarioPv.Intrnl.Edit_Scenario_Number,EditScenarioPv.Intrnl.Old_Scenario_Number)[OTE(EditScenarioPv.Ev.ScenarioNumberChanged) ,MOV(EditScenarioPv.Intrnl.Edit_Scenario_Number,EditScenarioPv.Intrnl.Old_Scenario_Number) ];
   23: NEQ(EditScenarioPv.Intrnl.Edit_Step_Number,EditScenarioPv.Intrnl.Old_Scenario_Step)[OTE(EditScenarioPv.Ev.StepNumberChanged) ,MOV(EditScenarioPv.Intrnl.Edit_Step_Number,EditScenarioPv.Intrnl.Old_Scenario_Step) ];
   24: XIC(EditScenario.Cmd.Accept_Configuration_Grid)[COP(EditScenarioPv.Intrnl.Scenario_Edit_Buffer.Output_Table.Data[0],Scenario[EditScenarioPv.Intrnl.Edit_Scenario_Number].Step[EditScenarioPv.Intrnl.Edit_Step_Number].Output_Table.Data[0],2) ,OTL(EditScenarioPv.Ev.Grid_Configuration_Accepted) ,OTU(EditScenario.Cmd.Accept_Configuration_Grid) ];
